FUNCTION_BLOCK FB_MedidorTapa_SFC // EXTENDS FB_Module_SFC
VAR_INPUT
	IC: BOOL;
	Execute: BOOL;
	Ack: BOOL;
END_VAR
VAR_OUTPUT
	Ready: BOOL;
	Failure: BOOL;
	Done: BOOL;
END_VAR
// TODO CAMBIAR EL SITIO DE RECOGER LA MEDIDA, NO ESPERAR A QUE SUBA EL MEDIDOR PARA RECOGER EL NÚMERO SINO QUE HACERLO JUSTO CUANDO TERMINE DE BAJAR
VAR_INPUT
	ctInp: S_ControllerInput;
	TMED: TIME := T#1S;			// Temporizador medición tapa
	fv: UINT; 					// Detector valor altura 
	LecturaFiable: BOOL;		// La lectura de la altura ha terminado 	
END_VAR

VAR_OUTPUT
	ctOut: S_ControllerOutput;
	L_1: BOOL; 					// Medidor de altura baja
	Leyendo: BOOL;
END_VAR

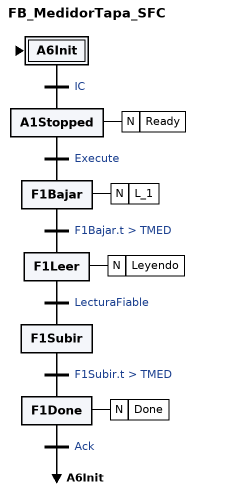
INITIAL_STEP A6Init:
END_STEP
TRANSITION FROM A6Init TO A1Stopped
    := IC;
END_TRANSITION
STEP A1Stopped:
    Ready(N);
END_STEP
TRANSITION FROM A1Stopped TO F1Bajar
    := Execute;
END_TRANSITION
STEP F1Bajar:
    L_1(N);
END_STEP
TRANSITION FROM F1Bajar TO F1Leer
    := F1Bajar.t > TMED;
END_TRANSITION
STEP F1Leer:
    Leyendo(N);
END_STEP
TRANSITION FROM F1Leer TO F1Subir
    := LecturaFiable;
END_TRANSITION
STEP F1Subir:
END_STEP
TRANSITION FROM F1Subir TO F1Done
    := F1Subir.t > TMED;
END_TRANSITION
STEP F1Done:
    Done(N);
END_STEP
TRANSITION FROM F1Done TO A6Init
    := Ack;
END_TRANSITION

END_FUNCTION_BLOCK

(* stored: Version 1.1.0.1, ProductVersion 3.1.4024.11
   POU FB_MedidorTapa_SFC: Id {586537d7-6cab-450b-b2b9-fb1352203f2f}, SpecialFunc None *)
